(* IEC 61131-3 sources: router_agent/data/raw-data/benchmark_raw/221_BottleProcessing/plc_st_files, 1 file *)

(* ---- 221_BottleProcessing.st ---- *)
FUNCTION_BLOCK FB_BottleProcessing
VAR_INPUT
    bottleSensor : BOOL; (* Sensor signal indicating a bottle is detected *)
    cleaningConfirmButton : BOOL; (* Operator button to confirm cleaning completion *)
    fillingConfirmButton : BOOL; (* Operator button to confirm filling completion *)
    cappingConfirmButton : BOOL; (* Operator button to confirm capping completion *)
    packingConfirmButton : BOOL; (* Operator button to confirm packaging completion *)
    finishedButton : BOOL; (* Operator button to confirm the bottle has been picked up *)
END_VAR
VAR_OUTPUT
    Pump_Motor : BOOL; (* Control output for the cleaning pump motor *)
    Filling_Valve : BOOL; (* Control output for the filling valve *)
    Capping_Machine : BOOL; (* Control output for the capping machine *)
    Packing_Machine : BOOL; (* Control output for the packing machine *)
    Completion_Light : BOOL; (* Indicator light for packaging completion *)
END_VAR
VAR
    cleaningStep : BOOL := FALSE;
    fillingStep : BOOL := FALSE;
    cappingStep : BOOL := FALSE;
    packingStep : BOOL := FALSE;
    completionStep : BOOL := FALSE;
END_VAR

IF bottleSensor THEN
    cleaningStep := TRUE;
    Pump_Motor := TRUE;
    Filling_Valve := FALSE;
    Capping_Machine := FALSE;
    Packing_Machine := FALSE;
    Completion_Light := FALSE;
END_IF;

IF cleaningConfirmButton AND cleaningStep THEN
    cleaningStep := FALSE;
    fillingStep := TRUE;
    Pump_Motor := FALSE;
    Filling_Valve := TRUE;
    Capping_Machine := FALSE;
    Packing_Machine := FALSE;
    Completion_Light := FALSE;
END_IF;

IF fillingConfirmButton AND fillingStep THEN
    fillingStep := FALSE;
    cappingStep := TRUE;
    Pump_Motor := FALSE;
    Filling_Valve := FALSE;
    Capping_Machine := TRUE;
    Packing_Machine := FALSE;
    Completion_Light := FALSE;
END_IF;

IF cappingConfirmButton AND cappingStep THEN
    cappingStep := FALSE;
    packingStep := TRUE;
    Pump_Motor := FALSE;
    Filling_Valve := FALSE;
    Capping_Machine := FALSE;
    Packing_Machine := TRUE;
    Completion_Light := FALSE;
END_IF;

IF packingConfirmButton AND packingStep THEN
    packingStep := FALSE;
    completionStep := TRUE;
    Pump_Motor := FALSE;
    Filling_Valve := FALSE;
    Capping_Machine := FALSE;
    Packing_Machine := FALSE;
    Completion_Light := TRUE;
END_IF;

IF finishedButton AND completionStep THEN
    cleaningStep := FALSE;
    fillingStep := FALSE;
    cappingStep := FALSE;
    packingStep := FALSE;
    completionStep := FALSE;
    Pump_Motor := FALSE;
    Filling_Valve := FALSE;
    Capping_Machine := FALSE;
    Packing_Machine := FALSE;
    Completion_Light := FALSE;
END_IF;

END_FUNCTION_BLOCK
